PROGRAM MAIN
VAR
END_VAR

END_PROGRAM

(* stored: Version 1.1.0.1
   POU MAIN: Id {8289c0cf-ec6a-42d4-bc96-7e3b0a802adb} *)
